// Mitsubishi GX Works2 project: tanque3   PLC: FX3U/FX3UC
// Configuração Modbus RTU

PROGRAM MAIN
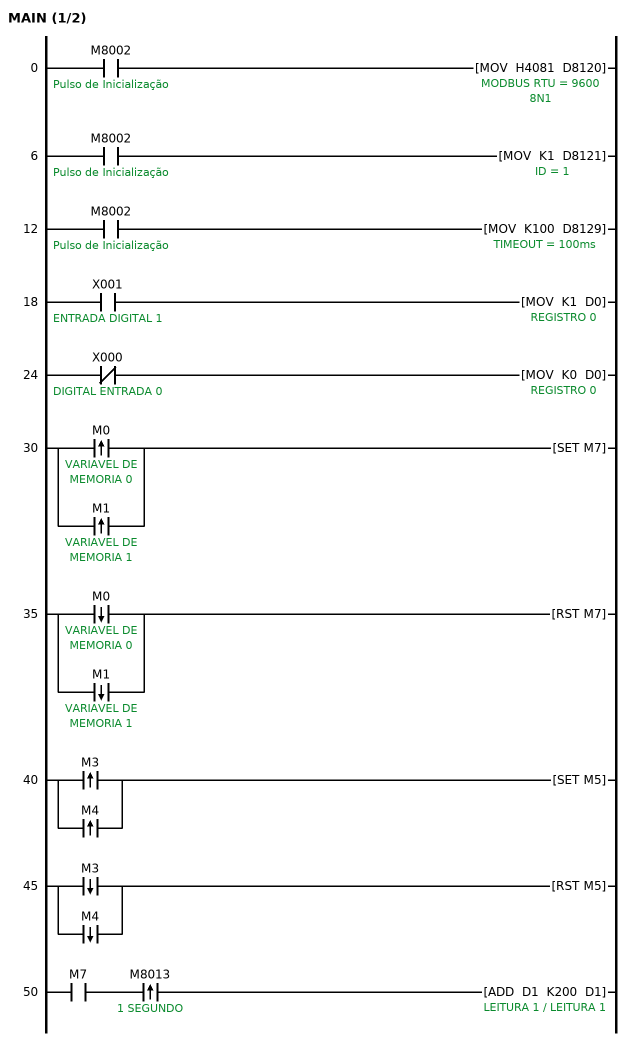
0     LD      M8002  ; Pulso de Inicialização
      MOV     H4081 D8120  ; MODBUS RTU = 9600 8N1
6     LD      M8002  ; Pulso de Inicialização
      MOV     K1 D8121  ; ID = 1
12    LD      M8002  ; Pulso de Inicialização
      MOV     K100 D8129  ; TIMEOUT = 100ms
18    LD      X001  ; ENTRADA DIGITAL 1
      MOV     K1 D0  ; REGISTRO 0
24    LDI     X000  ; DIGITAL ENTRADA 0
      MOV     K0 D0
30    LDP     M0  ; VARIAVEL DE MEMORIA 0
      ORP     M1  ; VARIAVEL DE MEMORIA 1
      SET     M7
35    LDF     M0  ; VARIAVEL DE MEMORIA 0
      ORF     M1  ; VARIAVEL DE MEMORIA 1
      RST     M7
40    LDP     M3
      ORP     M4
      SET     M5
45    LDF     M3
      ORF     M4
      RST     M5
50    LD      M7
      ANDP    M8013  ; 1 SEGUNDO
      ADD     D1 K200 D1  ; LEITURA 1
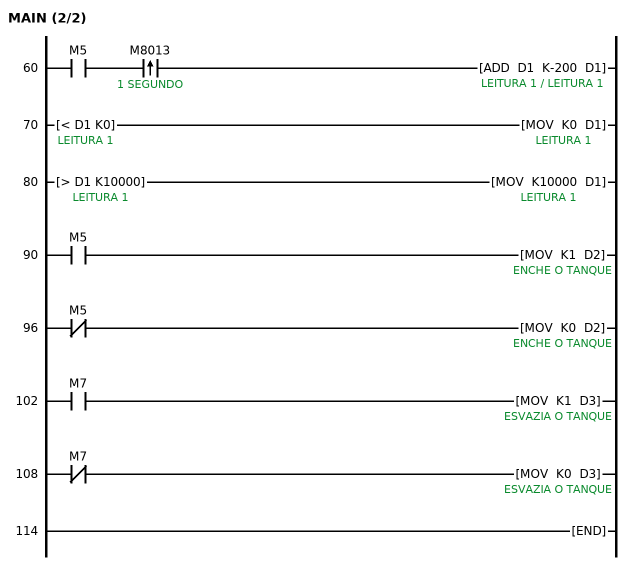
60    LD      M5
      ANDP    M8013  ; 1 SEGUNDO
      ADD     D1 K-200 D1
70    LD<     D1 K0  ; LEITURA 1
      MOV     K0 D1
80    LD>     D1 K10000  ; LEITURA 1
      MOV     K10000 D1
90    LD      M5
      MOV     K1 D2  ; ENCHE O TANQUE
96    LDI     M5
      MOV     K0 D2
102   LD      M7
      MOV     K1 D3  ; ESVAZIA O TANQUE
108   LDI     M7
      MOV     K0 D3
114   END
END_PROGRAM

// device comments not shown above
Y000  ; RELE 0
Y001  ; RELE 1
Y002  ; RELE 2
M2  ; VARIAVEL DE MEMORIA 2
